Fanuc KAREL source: kt00403.KL

-- PROVISIONAL review KL for V1013-1; original PC SHA256 3377b1fa44c34ac3a015efdb48d302a286c62a1afdbf7216b82701eb9a579b64
-- Incomplete behavior may be omitted. Consult companion uncertainty JSON. Do not deploy.
PROGRAM KT00403
%NOLOCKGROUP
VAR
  I1 : INTEGER
  OUT : BOOLEAN
-- UNRESOLVED_DECL Y2 type=002018
BEGIN
  -- UNRESOLVED_PC offsets 5-16; opcodes 2E,23
  -- UNRESOLVED_PC offsets 21-35; opcodes 2E,22,9D,33,B2
  -- UNRESOLVED_PC offsets 40-62; opcodes 21,22,9D,33,B1,5B,23
  -- UNRESOLVED_PC offsets 67-71; opcodes 7F
END KT00403
